PROGRAM PRG_TF3600_Math
VAR_INPUT
    fActualRPM : LREAL := 1000.0;
END_VAR

VAR CONSTANT
    cN          : UDINT := 2500;  
    cREF        : LREAL := 1000.0; 
    cFFT_LO     : UDINT := 1;      
    cFFT_HI     : UDINT := 250;    
    cLF_BINS    : UDINT := 3;      
    cALPHA      : LREAL := 11.3;   
    cCH         : UDINT := 6;     
    cSPEC_LEN   : UDINT := 250;    
END_VAR

VAR
    // --- Angular resampling ---
    fResampleRatio  : LREAL;                                             
    nResampledLen   : UDINT;                                             
    aResampled      : ARRAY[1..6, 0..2999] OF LREAL;                    
    fIdx            : LREAL;
    nIdx0, nIdx1    : UDINT;
    fFrac           : LREAL;

    // --- Hann window ---
    aHann           : ARRAY[0..2499] OF LREAL;
    aWindowed       : ARRAY[1..6, 0..2499] OF LREAL;
    bHannReady      : BOOL := FALSE;

    // --- FFT via TF3600 ---
    fbFFT           : ARRAY[1..6] OF FB_CMA_MagnitudeSpectrum;
    aFFTOut         : ARRAY[1..6, 0..1250] OF LREAL;                  
    aFFTIn          : ARRAY[0..2499] OF LREAL;                    

    // --- Log-magnitude spectrum ---
    aLogMag         : ARRAY[1..6, 0..249] OF LREAL;                    

    // --- Speed correction ---
    fLogR           : LREAL;                                             

    // --- Output ---
    aSpectrum       : ARRAY[0..1499] OF LREAL;

    // --- Loop indices ---
    ch, i, b        : UDINT;
    nFlatIdx        : UDINT;
END_VAR


IF NOT PRG_Slicer.bBufferReady THEN
    RETURN;
END_IF

// ── 1. Hann window ─────────────────────────────────────────────
IF NOT bHannReady THEN
    FOR i := 0 TO cN - 1 DO
        aHann[i] := 0.5 * (1.0 - COS(2.0 * LREAL_TO_LREAL(3.14159265358979) * INT_TO_LREAL(i) / INT_TO_LREAL(cN - 1)));
    END_FOR
    bHannReady := TRUE;
END_IF

// ── 2. Angular resampling  ──────────────────────────
fResampleRatio := fActualRPM / cREF;
nResampledLen  := LREAL_TO_UDINT(LREAL_TO_LREAL(cN) * fResampleRatio + 0.5);

FOR ch := 1 TO cCH DO
    FOR i := 0 TO nResampledLen - 1 DO
        // Map output index back to input index
        fIdx  := INT_TO_LREAL(i) * INT_TO_LREAL(cN - 1) / INT_TO_LREAL(nResampledLen - 1);
        nIdx0 := LREAL_TO_UDINT(fIdx);
        nIdx1 := nIdx0 + 1;
        fFrac := fIdx - INT_TO_LREAL(nIdx0);

        IF nIdx1 >= cN THEN
            nIdx1 := cN - 1;
        END_IF

        aResampled[ch, i] := PRG_Slicer.aWindowBuffer[ch, nIdx0 + 1, PRG_Slicer.nReadyBuffer] * (1.0 - fFrac)
                           + PRG_Slicer.aWindowBuffer[ch, nIdx1 + 1, PRG_Slicer.nReadyBuffer] * fFrac;
    END_FOR
END_FOR

// ── 3. Hann window ───────────
FOR ch := 1 TO cCH DO
    FOR i := 0 TO cN - 1 DO
        IF i < nResampledLen THEN
            aWindowed[ch, i] := aResampled[ch, i] * aHann[i];
        ELSE
            aWindowed[ch, i] := 0.0;
        END_IF
    END_FOR
END_FOR

// ── 4. FFT magnitude ─────────────────
FOR ch := 1 TO cCH DO
    FOR i := 0 TO cN - 1 DO
        aFFTIn[i] := aWindowed[ch, i];
    END_FOR

    fbFFT[ch](
        pDataIn      := ADR(aFFTIn),
        nDataInSize  := SIZEOF(aFFTIn),
        pDataOut     := ADR(aFFTOut[ch, 0]),
        nDataOutSize := SIZEOF(aFFTOut) / cCH,
        eWindowType  := eMA_WindowType_None,   // window already applied manually
        bExecute     := TRUE
    );
END_FOR

// ── 5. log1p of magnitude ───────────────────
FOR ch := 1 TO cCH DO
    FOR b := 0 TO cSPEC_LEN - 1 DO
        aLogMag[ch, b] := LN(1.0 + aFFTOut[ch, b + cFFT_LO]);
    END_FOR
END_FOR

// ── 6. Fixed-alpha speed correction ──────────────────────────────────────
fLogR := LN(fActualRPM / cREF);

FOR ch := 1 TO cCH DO
    FOR b := 0 TO cSPEC_LEN - 1 DO
        aLogMag[ch, b] := aLogMag[ch, b] - 2.0 * fLogR;
    END_FOR
    FOR b := 0 TO cLF_BINS - 1 DO
        aLogMag[ch, b] := aLogMag[ch, b] - (cALPHA - 2.0) * fLogR;
    END_FOR
END_FOR

// ── 7. Flatten ───────
nFlatIdx := 0;
FOR ch := 1 TO cCH DO
    FOR b := 0 TO cSPEC_LEN - 1 DO
        aSpectrum[nFlatIdx] := aLogMag[ch, b];
        nFlatIdx := nFlatIdx + 1;
    END_FOR
END_FOR


PRG_Slicer.bBufferReady := FALSE;

END_PROGRAM

(* stored: Version 1.1.0.1, ProductVersion 3.1.4024.15
   POU PRG_TF3600_Math: Id {dcba501c-a882-4848-9545-95becc9867c4}, SpecialFunc None *)
